# B&R Automation Studio project bms
Automation Studio 3.0.80.25; Default project

## Configuration MainStation

### Task classes (Cpu.sw)
```
Cyclic#1:
  hs_con <- MainStation.HeatingSystem.hs_con.prg
  ip_con <- MainStation.IrrigationSystem.ip_con.prg
  hmi_sup <- MainStation.hmi_sup.prg
Cyclic#2:
  rcp_cpy <- MainStation.rcp_cpy.prg
  alarm <- MainStation.alarm.prg
  statistics <- MainStation.statistics.prg
DataObjects: rcp_def <- MainStation.rcp_def.dob, arsdmsvp, arsdmsvg, arsdmhtm, heatcurv <- MainStation.HeatingSystem.heatcurv.dob, lin_heat <- MainStation.HeatingSystem.lin_heat.dob, lin_in <- MainStation.HeatingSystem.lin_in.dob, lin_out <- MainStation.HeatingSystem.lin_out.dob, temph_10, bms_stat, templ_08, temph05, heat_03, temph_05, heat_04, templ_07, templ_09, temph_09, heat_09, templ_06, heat_10, temph_07, templ_04, temph_02, templ_05, heat_05, templ_02, temph_03, templ05, temph_04, heat_02, templ_03, heat_06, heat_07, temph_06, templ_10, temph_08
VcDataObjects: MainHM <- MainStation.MainHMI.dob
Binaries: arsdm, webserv, vcmgr, vccbtn, vccshape, vcbclass, vcgclass, vcfile, vccnum, vccbmp, vcfntttf, vctcal, vcalarm, MainHM01, MainHM02, arial, vcresman, vcpdsw, vccovl, arialbd, vcchspot, visapi, vcshared, MainHM03, vcrt, vcctext, vcctrend, vcdsloc, vcdsint, vcchtml, vccalarm, vcclbox, vcxml, vccurl, vccbar, vccline, vcpfar00, vcnet, visvc, vcpdvnc, ashwd, sysconf, arconfig, iomap, asfw, PW3502, PW3501, vcinter, ddpccan, aplib, vcptelo, vcpdpp30, vcpfmtcx, vcpfpp30
Libraries: DataObj, astime, astcp, convert, asmem, runtime, sys_lib, fileio, bmslib, brsystem, loopconr, vcscrsht, asstring, can_lib
```

### IoMap.iom - PP420/IoMap.iom
```iecst
(********************************************************************
 * COPYRIGHT --
 ********************************************************************
 * File: IoMap.iom
 * Author: asdemo
 * Created: December 29, 2009
 ********************************************************************
 * IO mapping file
 ********************************************************************)
VAR_CONFIG
	diTankLevelHigh AT %IX.SL1.SS1.IF2.ST2.DigitalInput03;
	diTankLevelLow AT %IX.SL1.SS1.IF2.ST2.DigitalInput04;
	doIrrigValve1 AT %QX.SL1.SS1.IF2.ST2.DigitalOutput01; (*Rasenregner*)
	doIrrigValve2 AT %QX.SL1.SS1.IF2.ST2.DigitalOutput02; (*Beide Grander*)
	doIrrigValve3 AT %QX.SL1.SS1.IF2.ST2.DigitalOutput03; (*Gemüse - oben*)
	doIrrigValve4 AT %QX.SL1.SS1.IF2.ST2.DigitalOutput04; (*Gemüse - mitte*)
	doIrrigValve5 AT %QX.SL1.SS1.IF2.ST2.DigitalOutput05; (*Gemüse - unten*)
	doIrrigValve6 AT %QX.SL1.SS1.IF2.ST2.DigitalOutput06; (*Blumenhang*)
	doIrrigPump AT %QX.SL1.SS1.IF2.ST2.DigitalOutput08;
	aiTempBoiler AT %IW.SL1.SS1.IF2.ST3.SL1.SS1.Resistor01;
	aiTempBurner AT %IW.SL1.SS1.IF2.ST3.SL1.SS1.Resistor02;
	aiTempFlow AT %IW.SL1.SS1.IF2.ST3.SL1.SS1.Resistor03;
	aiTempOutside AT %IW.SL1.SS1.IF2.ST3.SL1.SS1.Resistor04;
	aiTempLivingroom AT %IW.SL1.SS1.IF2.ST3.SL1.SS2.Resistor01;
	doBurner AT %QX.SL1.SS1.IF2.ST3.SL2.DigitalOutput01;
	doFlowPump AT %QX.SL1.SS1.IF2.ST3.SL2.DigitalOutput02;
	doBoilerPump AT %QX.SL1.SS1.IF2.ST3.SL2.DigitalOutput03;
	doMixerOpen AT %QX.SL1.SS1.IF2.ST3.SL3.DigitalOutput01;
	doMixerClose AT %QX.SL1.SS1.IF2.ST3.SL3.DigitalOutput02;
	gIrrigationNodeOk AT %IX.SL1.SS1.IF2.ST2.ModuleOk;
	gHeatingNodeTemp1Ok AT %IX.SL1.SS1.IF2.ST3.SL1.SS1.ModuleOk;
	gHeatingNodeTemp2Ok AT %IX.SL1.SS1.IF2.ST3.SL1.SS2.ModuleOk;
	gHeatingNodeRelais1Ok AT %IX.SL1.SS1.IF2.ST3.SL2.ModuleOk;
	gHeatingNodeRelais2Ok AT %IX.SL1.SS1.IF2.ST3.SL3.ModuleOk;
END_VAR
```


## Logical view

Binary libraries used (declarations not repeated): astime, brsystem, DataObj, FileIO, LoopConR 2.71.2, sys_lib, VcScrSht, Visapi

### History.dat
```
08.05.2010:
- erste Installation, Inbetriebnahme

22.05.2010:
- automatische Übernahme der Reglerparameter
- Brenner-Solltemperatur auf 71°C begrenzen
- Legionellen-Temperatur auf 65°C
- Brenner-Alarm auf 85°C
- Brennerhysterese auf +0°C und -2°C
- Minimale Brennerlaufzeit auf 60000ms (1 min)
- Brenner bei Übertemperatur mit Boiler kühlen wenn (Boiler < 80°C)
- horizontale Gitternetzlinien für Tagestemperatur-Trend
- Color-Datenpunkt für Regler eingeschaltet korrigiert
- neue Mixer-Statemachine damit es nicht zum Flackern der I/Os kommt wenn nahe am Toleranzband

02.06.2010:
- updatePID immer wenn Heizung eingeschalten wird, da LCRslimPID die Reglerparameter verliert?
- Heizkurve im 10° und 15!° Bereich um ca. 5° angehoben

03.07.2010:
- Statemachine für Warmwasser-Heizung:
	- Scharf im Zeitfenster
	- Wenn Entscheidung getroffen -> heizen bis Temperatur erreicht
	- Boiler-Pumpe erst einschaltung wenn Brenner-Temperatur nur mehr 5° unter Boiler-Soll ist
	- bei Legionellenabtötung wird rcpPar-Parameter überladen
- Neue Reglereinstellungen: Kp = 4 statt 6, Tn = 200 stat 180
- tempFlowSetOffset wird auf 0 begrenzt um negative Temperature an heissen Tagen zu vermeiden
- Hotspots für Bewässerung neu angeordnet: Blumenhang verschoben, doppelter Hotspot für Grander
```

### notizen.dat
```
Erweiterungen:
- 2008er Aufzeichnungen vorhanden?
1. Kickinger Robert: Reglereinstellung
	- Tuning einer Wohnraum Heizung mit Heizkörper und Raumfühler?
2. Brennerstörung rücklesen über Anpassungsmodul auf AF101 -> neuer Alarm
```

- Visualisation Logical/Basement/PW35 (not shown)

### Global.var - Global variables
```iecst
(********************************************************************
 * COPYRIGHT --  WERNER PAULIN
 ********************************************************************
 * File: Global.var
 * Author: paulinw
 * Created: December 26, 2009
 ********************************************************************
 * Global variables of project bms
 ********************************************************************)
VAR RETAIN
	gActData : actData_typ; (*actual data of BMS*)
END_VAR
VAR
	gSimulation : simulation_typ := (0); (*simulation data*)
	gCfg : cfg_typ := (0); (*includes validated recipe date to be used in other programs*)
	gHMI : hmi_typ := (0); (*inculdes recipe data and other interface variables for HMI*)
	gIrrigationNodeOk : BOOL := FALSE; (*indicator whether IO node for irrigation is connected*)
	gHeatingNodeTemp1Ok : BOOL := FALSE; (*indicator whether IO node for heating is connected*)
	gHeatingNodeTemp2Ok : BOOL := FALSE; (*indicator whether IO node for heating is connected*)
	gHeatingNodeRelais1Ok : BOOL := FALSE; (*indicator whether IO node for heating is connected*)
	gHeatingNodeRelais2Ok : BOOL := FALSE; (*indicator whether IO node for heating is connected*)
END_VAR
VAR CONSTANT
	BMS_STATISTICS_DO_NAME : STRING[10] := 'bms_stat'; (*data object containing statistical data of BMS*)
	MAX_SEGMENT_INDEX : UINT := 5; (*maximum segment index*)
	MAX_HOTWATER_TIME_INDEX : UINT := 1; (*maximum time zone index for hot water schedule*)
	DO_NAME_TREND_HEAT : STRING[10] := 'heat_'; (*dataobject name of burner temperature logging*)
	DO_NAME_TREND_TEMP_HIGH : STRING[10] := 'temph_'; (*dataobject name of high temperature logging*)
	DO_NAME_TREND_TEMP_LOW : STRING[10] := 'templ_'; (*dataobject name of low temperature logging*)
	BURNER_MAX_SET_TEMP : REAL := 71.0; (*maximum allowed set value for temperature of burner*)
	BURNER_MAX_TEMP : REAL := 85.0; (*maximum allowed temperature of burner*)
	BOILER_MAX_TEMP : REAL := 80.0; (*maximum boiler temperature*)
	MAX_TREND_YEAR_INDEX : UINT := 1; (*maximum year trends*)
	MAX_SAMPLE_INDEX_YEAR : UINT := 365; (*maximum index of samples in a year*)
	MAX_SAMPLE_INDEX_DAY : UINT := 359; (*maximum samples in a day*)
	MAX_TREND_DAY_INDEX : UINT := 1; (*maximum day trends*)
END_VAR
```

### IO.var - Package variables
```iecst
(********************************************************************
 * COPYRIGHT --  WERNER PAULIN
 ********************************************************************
 * File: IO.var
 * Author: paulinw
 * Created: December 27, 2009
 ********************************************************************
 * Global variables of project bms
 ********************************************************************)
(*Irrigation sysem I/Os*)
VAR
	diTankLevelHigh : BOOL := FALSE; (*tank level indicator high*)
	diTankLevelLow : BOOL := FALSE; (*tank level indicator low*)
	doIrrigValve1 : BOOL := FALSE; (*valve on/off*)
	doIrrigValve2 : BOOL := FALSE; (*valve on/off*)
	doIrrigValve3 : BOOL := FALSE; (*valve on/off*)
	doIrrigValve4 : BOOL := FALSE; (*valve on/off*)
	doIrrigValve5 : BOOL := FALSE; (*valve on/off*)
	doIrrigValve6 : BOOL := FALSE; (*valve on/off*)
	doIrrigPump : BOOL := FALSE; (*valve on/off*)
END_VAR
(*Heating system I/Os*)
VAR
	aiTempBurner : UINT; (*raw value of temperature sensor: burner*)
	aiTempFlow : UINT; (*raw value of temperature sensor: flow temperature*)
	aiTempOutside : UINT; (*raw value of temperature sensor: outside*)
	aiTempLivingroom : UINT; (*raw value of temperature sensor: livingroom*)
	aiTempBoiler : UINT; (*raw value of temperature sensor: boiler*)
	doBurner : BOOL := FALSE; (*burner on/off*)
	doFlowPump : BOOL := FALSE; (*flow pump on/off*)
	doBoilerPump : BOOL := FALSE; (*boiler pump on/off*)
	doMixerOpen : BOOL := FALSE; (*open mixer*)
	doMixerClose : BOOL := FALSE; (*close mixer*)
END_VAR
```

### Alarms.typ - Package data types
```iecst
(********************************************************************
 * COPYRIGHT --
 ********************************************************************
 * File: Alarms.typ
 * Author: paulinw
 * Created: December 26, 2009
 ********************************************************************
 * Global data types of project bms
 ********************************************************************)
(*How to add new alarms:*)
(*1. add alarm in enum list*)
(*2. define reaction in alarm.st*)
(*3. add alarm in Visual Components*)
(*4. use the alarm in program*)

TYPE
	ALARMS :
		(
		ALARM_RECIPE_READ := 0,
		ALARM_RECIPE_WRITE,
		ALARM_RECIPE_NAME_INV,
		ALARM_HEATING_BURNER_TEMP_HIGH,
		ALARM_HEATING_BOILER_TEMP_HIGH,
		ALARM_HEATING_NODE_CON_ERROR,
		ALARM_IRRIGATION_NODE_CON_ERROR,
		ALARM_HEATING_BURNER_TEMP_LIMIT,
		ALARM_MAX
		);
	ALARM_REACTIONS :
		(
		ALARM_REACTION_NOTHING := 0,
		ALARM_REACTION_STOP,
		ALARM_REACTION_WARNING
		);
	alarm_typ : 	STRUCT
		request : ARRAY[0..ALARM_MAX] OF BOOL;
		ack : ARRAY[0..ALARM_MAX] OF BOOL;
		reaction : ARRAY[0..ALARM_MAX] OF DINT;
		warning : BOOL;
		stop : BOOL;
		ackBlock : BOOL;
	END_STRUCT;
END_TYPE
```

### Alarms.var - Package variables
```iecst
(********************************************************************
 * COPYRIGHT --
 ********************************************************************
 * File: Alarms.var
 * Author: paulinw
 * Created: December 26, 2009
 ********************************************************************
 * Global variables of project bms
 ********************************************************************)
VAR
	gAlarm : alarm_typ := (0); (*alarm data*)
END_VAR
VAR CONSTANT
	NB_ALARMS : ALARMS := ALARM_MAX;
END_VAR
```

### Library Logical/Libraries/bmslib (IEC)

#### bmslib.st
```iecst
(********************************************************************
 * COPYRIGHT -- WERNER PAULIN
 ********************************************************************
 * Package: bmslib
 * File: bmslib.st
 * Author: paulinw
 * Created: December 27, 2009
 *******************************************************************)

(* writes data to dataobjects and creates it if it does not exists *)
FUNCTION_BLOCK DatObjUpdate
	fDatObjInfo(enable := 1, pName := pName);

	(* create data object if it does not exists *)
	IF (fDatObjInfo.status <> ERR_OK) OR (fDatObjCreate.status = ERR_FUB_BUSY) THEN
		fDatObjCreate(enable := 1, grp := 0, pName := fDatObjInfo.pName, len := nbElement * sizeOfElement, MemType := doUSRROM, Option := 0, pCpyData := 0);

		IF (fDatObjCreate.status = ERR_FUB_BUSY) THEN		(* wait until fub is finished *)
			status := ERR_FUB_BUSY;
			RETURN;
		ELSIF (fDatObjCreate.status = ERR_OK) THEN			(* save ident for writing if finished without error *)
  			ident := fDatObjCreate.ident;
   		ELSE												(* return any error and abort fub *)
			status := fDatObjCreate.status;
			RETURN;
		END_IF;
	ELSIF (fDatObjInfo.status = ERR_OK) THEN				(* save ident for writing if finished without error *)
		ident := fDatObjInfo.ident;
	END_IF;

	(* start writing only if module was created or found *)
	IF (ident <> 0) THEN
		fDatObjWrite(enable := 1, ident := ident, Offset := index * sizeOfElement, pSource := pData, len := sizeOfElement);
		status := fDatObjWrite.status;
		RETURN;
	END_IF;

	status := ERR_FUB_BUSY;
END_FUNCTION_BLOCK

(* Irrigation Valve Manager *)
FUNCTION_BLOCK IrrigValveMgr
	(* monitor ontime with watch in order to avoid that user forgets to switch off segment *)
	IF (switchOnRequest = TRUE) THEN
		watchdogTimer := watchdogTimer + newMinute;
		IF (watchdogTimer >= SEGMENT_WATCHDOG_TIME) THEN
			switchOnRequest := FALSE;
			watchdogTimer := 0;
  		END_IF;
	ELSE
		watchdogTimer := 0;
	END_IF;

	pumpRequest := valve := switchOnRequest;		(* switch on valve and request pump to be switched on *)
END_FUNCTION_BLOCK

(* calculates the day of a year from a date *)
FUNCTION DayOfYear
	(* plausibility *)
	IF (inDate.month = 0) OR (inDate.month > 12) OR (inDate.day = 0) OR (inDate.day > 31) THEN
		DayOfYear := 1;
		RETURN;
	END_IF;

	(* count all days before this month *)
	DayOfYear := 0;
	FOR monthIndex := 1 TO inDate.month-1 DO
		DayOfYear := DayOfYear + dayPerMonth[monthIndex];
	END_FOR;

	(* add days of current month *)
	DayOfYear := DayOfYear + inDate.day;

	(* if year is a leap year and february has been already passed -> add one day because OF 29th OF feb. *)
	IF (IsLeapYear(inDate.year) = TRUE) AND (inDate.month > 2) THEN
		DayOfYear := DayOfYear + 1;
	END_IF;

	(* avoid invalid output *)
	IF (DayOfYear = 0) THEN
		DayOfYear := 1;
	END_IF;
END_FUNCTION

(* determine whether the given year is a leap year *)
FUNCTION IsLeapYear
	IF (((year MOD 4) = 0) AND ((year MOD 100) <> 0)) OR ((year MOD 400) = 0) THEN
		IsLeapYear := TRUE;
	ELSE
		IsLeapYear := FALSE;
	END_IF;
END_FUNCTION

(* 2 point hysteresis - optimized for heating *)
FUNCTION_BLOCK Hyst2p
	(* deviation: not used in function block but might be interesting for further usage *)
	e := xSet - xAct;

	(* switch off if temperature is outside of higher threshold *)
	IF (xAct > (xSet + pHyst)) THEN
		y := FALSE;
		xActOld := xAct;
	(* switch off if temperature has not yet reached lower threshold *)
	ELSIF ((xActOld > xAct) AND (xAct >= (xSet - nHyst))) THEN
		y := FALSE;
	(* switch on if temperature reached lower threshold *)
	ELSIF (xAct < (xSet - nHyst)) THEN
		y := TRUE;
		xActOld := xAct;
	ELSE
		y := TRUE;
	END_IF;
END_FUNCTION_BLOCK

(* Generates the name of a trend data object with the year in the suffix *)
FUNCTION_BLOCK GetTrendDatObjName
	memset(ADR(datObjName), 0, SIZEOF(datObjName));
	strcpy(ADR(datObjName), ADR(templateName));					(* template name *)

	itoa((year / 10) MOD 10, ADR(stringDigit));					(* add second digit of year *)
	strcat(ADR(datObjName), ADR(stringDigit));

	itoa((year /  1) MOD 10, ADR(stringDigit));					(* add first digit of year *)
	strcat(ADR(datObjName), ADR(stringDigit));
END_FUNCTION_BLOCK

(* calculates day and month according to a given day of year *)
FUNCTION_BLOCK DateOfDay
	(* plausibility *)
	IF (dayOfYear = 0) OR (dayOfYear > 366) THEN
		outDate.month := 1;
		outDate.day   := 1;
		RETURN;
	END_IF;

	(* adjust February in case of leap year *)
	IF IsLeapYear(year) = TRUE THEN
		dayPerMonth[2] := 29;
	ELSE
		dayPerMonth[2] := 28;
	END_IF;

	(* find month of this year's day *)
	dayOfYearSum := 0;
	FOR monthIndex := 1 TO 12 DO
		dayOfYearSum := dayOfYearSum + dayPerMonth[monthIndex];
		(* stop counting up days if desired day reached -> monthIndex shows the corresponding month *)
		IF dayOfYearSum >= dayOfYear THEN
			EXIT;
		END_IF;
	END_FOR;

	outDate.month := monthIndex;
	outDate.day   := dayPerMonth[monthIndex] - UINT_TO_USINT(dayOfYearSum - dayOfYear);		(* add the remaining days of this month *)
END_FUNCTION_BLOCK
```

### Package Logical/MainStation/HeatingSystem - Heating System Control

### Program Logical/MainStation/HeatingSystem/hs_con (IEC) - heating system controller

#### hs_con.var - Local variables
```iecst
(********************************************************************
 * COPYRIGHT --
 ********************************************************************
 * Program: hs_con
 * File: hs_con.var
 * Author: asdemo
 * Created: December 27, 2009
 ********************************************************************
 * Local variables of program hs_con
 ********************************************************************)
VAR
	fHyst2pBurner : Hyst2p;
	fHyst2pLivingRoom : Hyst2p;
	fGetTrendDatObjNameHighTemp : GetTrendDatObjName;
	fGetTrendDatObjNameLowTemp : GetTrendDatObjName;
	fLCRCurveByPoints : LCRCurveByPoints;
	index : UINT;
	minRuntimeTimerBurner : UDINT;
	fLCRSlimPID : LCRSlimPID;
	fRTInfo : RTInfo;
	dayMinute : UDINT;
	dmyTabEntry : lcrCurveByPoints_TabEntry_type;
	cntLoadOld : USINT;
	cycT : UDINT;
	fDatObjInfo : DatObjInfo;
	fDatObjUpdateYearTempLow : DatObjUpdate;
	fGetTrendDatObjNameHeat : GetTrendDatObjName;
	fDatObjUpdateYearHeat : DatObjUpdate;
	fDatObjUpdateYearTempHigh : DatObjUpdate;
	mixerRefTime : UDINT;
	pHeatCurve : UDINT;
	pLinDataInsideSensor : UDINT;
	oldMinute : USINT;
	nbPointsOutsideSensorLin : UINT;
	newMinute : BOOL;
	pLinDataOutsideSensor : UDINT;
	tempPIDrequest : UDINT;
	yearDay : UDINT;
	tempLCRSlimPIDpara : lcrslimpid_par_typ;
	rcpData : rcpData_typ;
	sStepMixer : REAL;
	nbPointsHeatCurve : UINT;
	pLinDataHeatSensor : UDINT;
	mixerRefTimer : UDINT;
	nbPointsInsideSensorLin : UINT;
	nbPointsHeatSensorLin : UINT;
	trendDebug : trendDebug_typ := (0);
END_VAR
VAR CONSTANT
	BMS_LIN_INSIDE_DO_NAME : STRING[10] := 'lin_in'; (*linearisation of inside temperature sensors*)
	BMS_LIN_HEAT_DO_NAME : STRING[10] := 'lin_heat'; (*linearisation of heating sensors*)
	BURNER_TEMP_SET_OFFSET : REAL := 5.0; (*Offset to set temperature to make sure heat is transported away from the burner*)
	BMS_HEATING_CURVE : STRING[10] := 'heatcurv'; (*relation between outside temperature and flow temperature*)
	BURNER_TEMP_POS_HYSTERESIS : REAL := 0.0; (*tolerance of burner temperature*)
	BURNER_TEMP_NEG_HYSTERESIS : REAL := 2.0; (*tolerance of burner temperature*)
	BURNER_PARALLEL_RESISTANCE : REAL := 4696.8; (*exact value of parallel restance used with NTC*)
	BURNER_MIN_RUNTIME : UDINT := 60000; (*minimum runtime of burner once switch on in ms*)
	HOTWATER_TEMP_LEGION_DISTINCTION : REAL := 65.0; (*hotwater set temperature for legionella distinction*)
	BMS_LIN_OUTSIDE_DO_NAME : STRING[10] := 'lin_out'; (*linearisation of outside temperature sensors*)
	BOILER_PARALLEL_RESISTANCE : REAL := 4715.8; (*exact value of parallel restance used with NTC*)
	LIVING_ROOM_TEMP_NEG_HYSTERESIS : REAL := 0.1; (*negative tolerance for living room temperature*)
	INSIDE_PARALLEL_RESISTANCE : REAL := 4651.1; (*exact value of parallel restance used with NTC*)
	LIVING_ROOM_TEMP_POS_HYSTERESIS : REAL := 0.3; (*positive tolerance for living room temperature*)
	MIXER_FULLY_OPEN_TIME : REAL := 118.0; (*time it takes to open the mixer fully*)
	MIXER_FULLY_OPEN_POSITION : REAL := 100.0; (*maximum position of mixer*)
	MIXER_ZERO_WINDOW : REAL := 0.9; (*don't move the mixer within this window in order to avoid lag errors*)
	CRITICAL_FREEZING_OUTSIDE_TEMP : REAL := 2.0; (*below this temperature heating water pipes may freeze on spots close to outside walls*)
	PID_HEATING_I_MAX : REAL := 100.0; (*anti windup of heating PID controller*)
	FLOW_PARALLEL_RESISTANCE : REAL := 4649.0; (*exact value of parallel restance used with NTC*)
	OUTSIDE_PARALLEL_RESISTANCE : REAL := 4692.2; (*exact value of parallel restance used with NTC*)
END_VAR
VAR
	fDatObjUpdateTempDebug : DatObjUpdate;
	fDatObjUpdateHeatDebug : DatObjUpdate;
	sMixer : UINT;
END_VAR
VAR CONSTANT
	sMIXER_STANDBY : UINT := 0;
	sMIXER_REFERENCE : UINT := 30;
	sMIXER_OPEN : UINT := 10;
	sMIXER_CLOSE : UINT := 20;
END_VAR
VAR
	oldHeatingEnable : BOOL;
	sHotwater : UINT;
END_VAR
VAR CONSTANT
	sHOTWATER_STANDBY : UINT := 0;
	sHOTWATER_WAIT_BURNER_HOT : UINT := 10;
	sHOTWATER_WAIT_HOTWATER_READY : UINT := 20;
END_VAR
```

#### hs_con.typ - Local data types
```iecst
(********************************************************************
 * COPYRIGHT -- Bernecker + Rainer
 ********************************************************************
 * Program: hs_con
 * File: hs_con.typ
 * Author: paulinw
 * Created: February 04, 2010
 ********************************************************************
 * Local data types of program hs_con
 ********************************************************************)

TYPE
	trendDebug_typ : 	STRUCT
		name : ARRAY[0..9] OF USINT;
		dayOfYear : UINT;
		date : DTStructure;
		dayOfYearFromDate : UINT;
		tempAct : REAL;
		tempSet : REAL;
		cmdTempSet : USINT;
		heatingHoursDayAct : UDINT;
		heatingHoursDaySet : UDINT;
		cmdHeatingHoursDaySet : USINT;
	END_STRUCT;
END_TYPE
```

### Program Logical/MainStation/HeatingSystem/hs_sim (IEC) - simulation of heating system

#### hs_sim.var
```iecst
(********************************************************************
 * COPYRIGHT --
 ********************************************************************
 * Program: hs_sim
 * File: hs_sim.var
 * Author: asdemo
 * Created: December 30, 2009
 ********************************************************************
 * Local variables of program hs_sim
 ********************************************************************)
VAR
	fLCRPT2burner : LCRPT2;
	fLCRPT2boiler : LCRPT2;
	fLCRPT2livingroom : LCRPT2;
	mixerBurner : REAL;
	mixerBackFlow : REAL;
	tempBackFlow : REAL;
	fLCRPT2flow : LCRPT2;
END_VAR
VAR CONSTANT
	SIM_ROOM_TEMP : REAL := 20.0;
END_VAR
```

### Data object Logical/MainStation/HeatingSystem/heatcurv (Simple)

#### heatcurv.dat
```
;+-----------------	outside temperature in °C (x-axis)
;|
;|     +----------- flow temperature in °C (y-axis)
;|     |
-20.0, 64.0
-15.0, 62.0
-10.0, 60.0
 -5.0, 59.0
  0.0, 58.0
  5.0, 57.0
 10.0, 55.0
 15.0, 50.0
 20.0, 32.0
```

- Data object Logical/MainStation/HeatingSystem/lin_heat (Simple) (no source held here)

- Data object Logical/MainStation/HeatingSystem/lin_in (Simple) (no source held here)

### Data object Logical/MainStation/HeatingSystem/lin_out (Simple)

#### lin_out.dat
```
; characteristic of outside temperature sensors

;+-------------------- resistance in Ohm (x-axis)
;|
;|        +----------- temperature in ?C (y-axis)
;|        |
 16000.0,  15.0,
 19000.0,  10.0,
 25000.0,   5.0,
 33000.0,   0.0,
 42000.0,  -5.0,
 55000.0, -10.0,
 76000.0, -15.0,
```

### Package Logical/MainStation/IrrigationSystem - Irrigation System Control

### Program Logical/MainStation/IrrigationSystem/ip_con (IEC) - irrigation plant controller

#### ip_con.var
```iecst
(********************************************************************
 * COPYRIGHT --
 ********************************************************************
 * Program: ip_con
 * File: ip_con.var
 * Author: asdemo
 * Created: December 27, 2009
 ********************************************************************
 * Local variables of program ip_con
 ********************************************************************)
VAR
	cycT : UDINT;
	fRTInfo : RTInfo;
	oldMinute : USINT;
	newMinute : BOOL;
	rcpData : rcpData_typ;
	IrrigValveMgr1 : IrrigValveMgr;
	IrrigValveMgr2 : IrrigValveMgr;
	IrrigValveMgr3 : IrrigValveMgr;
	IrrigValveMgr4 : IrrigValveMgr;
	IrrigValveMgr5 : IrrigValveMgr;
	IrrigValveMgr6 : IrrigValveMgr;
END_VAR
```

#### ip_con.st
```iecst
(********************************************************************
 * COPYRIGHT -- WERNER PAULIN
 ********************************************************************
 * Program: ip_con
 * File: ip_con.st
 * Author: paulinw
 * Created: December 27, 2009
 ********************************************************************
 * Implementation of program ip_con
 * Features:
 * - controlling 6 valves (fixed) and 1 pump
 * Interfaces:
 * - gActData.irrigation
 ********************************************************************
 * History:
 * Version	Date		Author		Comment
 * V1.00	27.12.09	W. Paulin	created
 ********************************************************************)

PROGRAM _INIT
	fRTInfo(enable := 1);
	cycT := fRTInfo.cycle_time / 1000;
END_PROGRAM

PROGRAM _CYCLIC
	(* generate flag indicating new minute *)
	IF (oldMinute <> gActData.general.time.minute) THEN
		newMinute := TRUE;
		oldMinute := gActData.general.time.minute;
	ELSE
		newMinute := FALSE;
	END_IF;

	(* apply recipe parameter if allowed  *)
	IF (gCfg.isValid) THEN
		memcpy(ADR(rcpData), ADR(gCfg.data), SIZEOF(rcpData));
	END_IF;

	(* link switches to valves including watchdog monitoring *)
	IrrigValveMgr1(newMinute := newMinute, switchOnRequest := gActData.irrigation.segment[0].switchOnRequest, valve := doIrrigValve1);
	IrrigValveMgr2(newMinute := newMinute, switchOnRequest := gActData.irrigation.segment[1].switchOnRequest, valve := doIrrigValve2);
	IrrigValveMgr3(newMinute := newMinute, switchOnRequest := gActData.irrigation.segment[2].switchOnRequest, valve := doIrrigValve3);
	IrrigValveMgr4(newMinute := newMinute, switchOnRequest := gActData.irrigation.segment[3].switchOnRequest, valve := doIrrigValve4);
	IrrigValveMgr5(newMinute := newMinute, switchOnRequest := gActData.irrigation.segment[4].switchOnRequest, valve := doIrrigValve5);
	IrrigValveMgr6(newMinute := newMinute, switchOnRequest := gActData.irrigation.segment[5].switchOnRequest, valve := doIrrigValve6);

	(* switch on pump if any valve requests water *)
	doIrrigPump := IrrigValveMgr1.pumpRequest OR
				   IrrigValveMgr2.pumpRequest OR
				   IrrigValveMgr3.pumpRequest OR
				   IrrigValveMgr4.pumpRequest OR
				   IrrigValveMgr5.pumpRequest OR
				   IrrigValveMgr6.pumpRequest;

	(* service cycle in order to void that valves get stuch during winter season *)
	IF (gActData.general.time.wday = 1) AND 		(* sunday to monday *)
	   (gActData.general.time.hour = 0) AND 		(* midnight *)
	   (doIrrigPump = FALSE) THEN					(* only if pump is switch off *)

		(* use valve outputs directly in order to avoid that pump will be switched on *)
		doIrrigValve1 := FALSE;
		doIrrigValve2 := FALSE;
		doIrrigValve3 := FALSE;
		doIrrigValve4 := FALSE;
		doIrrigValve5 := FALSE;
		doIrrigValve6 := FALSE;

		CASE gActData.general.time.minute OF		(* turn on every minute another valve *)
			1 : doIrrigValve1 := TRUE;
			2 : doIrrigValve2 := TRUE;
			3 : doIrrigValve3 := TRUE;
			4 : doIrrigValve4 := TRUE;
			5 : doIrrigValve5 := TRUE;
			6 : doIrrigValve6 := TRUE;
		END_CASE;
	END_IF;

	(* statistics *)
	gActData.statistics.irrigation.valve[0] := gActData.statistics.irrigation.valve[0] + EDGEPOS(doIrrigValve1);
	gActData.statistics.irrigation.valve[1] := gActData.statistics.irrigation.valve[1] + EDGEPOS(doIrrigValve2);
	gActData.statistics.irrigation.valve[2] := gActData.statistics.irrigation.valve[2] + EDGEPOS(doIrrigValve3);
	gActData.statistics.irrigation.valve[3] := gActData.statistics.irrigation.valve[3] + EDGEPOS(doIrrigValve4);
	gActData.statistics.irrigation.valve[4] := gActData.statistics.irrigation.valve[4] + EDGEPOS(doIrrigValve5);
	gActData.statistics.irrigation.valve[5] := gActData.statistics.irrigation.valve[5] + EDGEPOS(doIrrigValve6);

	IF (doIrrigPump = TRUE) THEN
		gActData.statistics.irrigation.onTimePump := gActData.statistics.irrigation.onTimePump + newMinute;
	END_IF;

	(* tank level feedback *)
	IF (diTankLevelHigh = TRUE) AND (diTankLevelLow = TRUE) THEN
		gActData.irrigation.tankLevel := 9;
	ELSIF (diTankLevelHigh = FALSE) AND (diTankLevelLow = TRUE) THEN
		gActData.irrigation.tankLevel := 6;
	ELSE
		gActData.irrigation.tankLevel := 3;
	END_IF;

	(* alarm handling *)
	gAlarm.request[ALARM_IRRIGATION_NODE_CON_ERROR] := NOT(gIrrigationNodeOk);
END_PROGRAM
```

### Data object Logical/MainStation/rcp_def (Simple) - default receipe

#### rcp_def.dat
```
(********************************************************************
 * COPYRIGHT -- WERNER PAULIN
 ********************************************************************
 * Data object: rcp_def
 * File: rcp_def.dat
 * Author: paulinw
 * Created: December 26, 2009
 ********************************************************************
 * Data object file: rcp_def.dat
 ********************************************************************
 * History:
 * Version	Date		Author		Comment
 * V1.00	26.12.10	W. Paulin	created
 ********************************************************************)
(* IMPORTANT: MAINTAIN 32bit ALIGNMENT!!! *)
; HEATING SYSTEM
0000000360, ; rcpData_typ.heating.startTime						/* (UDINT)   start time of heating [min] */
0000001350, ; rcpData_typ.heating.endTime						/* (UDINT)   end time of heating [min]   */
0000000001, ; rcpData_typ.heating.outOfHome.startDay			/* (UDINT)   out of home begin [day]     */
0000000002, ; rcpData_typ.heating.outOfHome.endDay				/* (UDINT)   out of home end [day]     */
20.0,       ; rcpData_typ.heating.tempLivingroomSet				/* (REAL)    living room set temperature [?C]  */
00.0,       ; rcpData_typ.heating.tempManOffset					/* (REAL)    manual offset to living room set temperature [°C] */
-2.0,       ; rcpData_typ.heating.tempLowOffset					/* (REAL)    lowering offset to living room set temperature [°C] */
0.0,		; rcpData_typ.heating.tempFlowSetOffset				/* (REAL)    offset to flow set temperature [°C] */
04.0,       ; rcpData_typ.heating.kp							/* (REAL)    kp of heating controller */
200.0,      ; rcpData_typ.heating.tn							/* (REAL)    tn of heating controller */
; HOT WATER
0000000450, ; rcpData_typ.heating.hotwater.startTime[0]			/* (UDINT)   start time of hot water [min] */
0000000990, ; rcpData_typ.heating.hotwater.startTime[1]			/* (UDINT)   start time of hot water [min] */
0000000480, ; rcpData_typ.heating.hotwater.endTime[0]			/* (UDINT)   start time of hot water [min] */
0000001050, ; rcpData_typ.heating.hotwater.endTime[1]			/* (UDINT)   start time of hot water [min] */
60.0,       ; rcpData_typ.heating.hotwater.tempSet				/* (REAL)    boiler set temperature [?C]  */
; IRRIGATION PLANT
; tbd...
```

### Program Logical/MainStation/rcp_cpy (IEC) - Receipe Handling

#### rcp_cpy.var
```iecst
(********************************************************************
 * COPYRIGHT --
 ********************************************************************
 * Program: rcp_cpy
 * File: rcp_cpy.var
 * Author: paulinw
 * Created: December 26, 2009
 ********************************************************************
 * Local variables of program rcp_cpy
 ********************************************************************)
VAR
	RECIPE_FILE_NAME_1 : STRING[10] := 'konfig_1';
	RECIPE_FILE_NAME_2 : STRING[10] := 'konfig_2';
	fDatObjInfo : DatObjInfo;
	fDatObjRead : DatObjRead;
	index : UINT;
	fDatObjUpdate : DatObjUpdate;
	actPicOld : UINT;
	newPage : BOOL;
END_VAR
VAR CONSTANT
	OK_FLAG_INVISIBLE : USINT := 0;
	OK_FLAG_ERROR : USINT := 2;
	OK_FLAG_OK : USINT := 1;
END_VAR
```

### Program Logical/MainStation/hmi_sup (IEC) - HMI support

#### hmi_sup.var - Local variables
```iecst
(********************************************************************
 * COPYRIGHT --
 ********************************************************************
 * Program: hmi_sup
 * File: hmi_sup.var
 * Author: asdemo
 * Created: December 27, 2009
 ********************************************************************
 * Local variables of program hmi_sup
 ********************************************************************)
VAR
	yearIndex : UINT;
	tempOutsideActOld : REAL;
	tempLivingroomActOld : REAL;
END_VAR
VAR CONSTANT
	TEMP_TENDENCY_UP : USINT := 1; (*temperature is rising*)
	TEMP_TENDENCY_HYSTERESIS : REAL := 0.1; (*hysteresis for temperature tendency generation*)
	TEMP_TENDENCY_DOWN : USINT := 0; (*temperature is falling*)
	sWAIT_CMD : UINT := 0;
END_VAR
VAR
	status : UDINT;
	sScrSht : UINT;
END_VAR
VAR CONSTANT
	sDO_SCREEN_SHOT : UINT := 10;
	sDEINIT : UINT := 20;
END_VAR
VAR
	pagePowerUpTimer : UDINT;
END_VAR
(* PAGE_HS_DIAG : USINT := 12; *)
(* PAGE_IS_OVERVIEW : USINT := 20; *)
(* PAGE_HS_CFG : USINT := 11; *)
VAR CONSTANT
	PAGE_POWERUP : USINT := 0; (*page: power up*)
	PAGE_SCREEN_CLEAN : USINT := 1;
	PAGE_BMS_CFG : USINT := 2;
	PAGE_HS_OVERVIEW : USINT := 10; (*page: heating system overview*)
END_VAR
VAR CONSTANT
	ONE_DAY : TIME := T#86400000ms; (*one day in milliseconds*)
END_VAR
VAR
	oldMinute : USINT;
	newPage : BOOL;
	newMinute : BOOL;
	nbDays : UINT;
	hScrSht : UDINT;
	fRTInfo : RTInfo;
	fileScrSht : STRING[10];
	fGetTrendDatObjName : GetTrendDatObjName;
	fDTStructureSetTime : DTStructureSetTime;
	fDTStructureGetTime : DTStructureGetTime;
	fDTGetTime : DTGetTime;
	fDatObjInfo : DatObjInfo;
END_VAR
VAR CONSTANT
	DELAY_POWERUP_PAGE : UINT := 1500; (*time delay to switch from power up page to heating system overview*)
END_VAR
VAR
	dayIndex : UINT;
	cycT : UDINT;
	cmdNewPageOld : UINT;
	actPicOld : UINT;
	bufferElementREAL : REFERENCE TO ARRAY[0..365] OF REAL;
	bufferElementUDINT : REFERENCE TO ARRAY[0..365] OF UDINT;
	cntMinute : USINT;
	new4Minute : BOOL;
END_VAR
VAR CONSTANT
	YESTERDAY : USINT := 0; (*buffer index containing data of yesterday*)
	TODAY : USINT := 1; (*buffer index containing data of today*)
END_VAR
VAR
	fDateOfDay : DateOfDay;
	index : UINT;
END_VAR
VAR CONSTANT
	SCREEN_CLEAN_TIME : UDINT := 30000;
END_VAR
VAR
	screenCleanTimer : UDINT;
	pageBeforeScreenClean : UINT;
	ledControl : ARRAY[0..5] OF USINT;
END_VAR
```

### Program Logical/MainStation/statistics (IEC) - statistical processing

#### statistics.var
```iecst
(********************************************************************
 * COPYRIGHT --
 ********************************************************************
 * Program: statistics
 * File: statistics.var
 * Author: asdemo
 * Created: December 27, 2009
 ********************************************************************
 * Local variables of program statistics
 ********************************************************************)
VAR
	fDatObjInfo : DatObjInfo;
	oldHour : USINT;
	cmdWriteStatistics : BOOL;
	fDatObjUpdate : DatObjUpdate;
	fDatObjRead : DatObjRead;
END_VAR
```

- Visualisation Logical/MainStation/MainHMI (not shown)

Listed in the project but not available here: Logical/Globals/Global.typ, Logical/Libraries/bmslib/bmslib.typ, Logical/Libraries/bmslib/bmslib.var, Logical/Libraries/bmslib/bmslib.fun, Logical/MainStation/HeatingSystem/hs_con/hs_con.st, Logical/MainStation/alarm, Logical/MainStation/hmi_sup/hmi_sup.st
